FUNCTION_BLOCK basicFalhaFeedbackOnOff (* Basic Function Block Type *)
  (* Standard: 61499-2 *)
  (* Version 0.0, 1/26/2026, Schneider Electric, Template *)
  PACKAGE Hidryco.HidrycoLib;
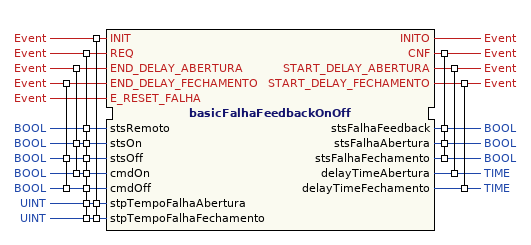
  EVENT_INPUT
    INIT WITH stpTempoFalhaAbertura, stpTempoFalhaFechamento; (* Initialization Request *)
    REQ WITH stsRemoto, stpTempoFalhaAbertura, stpTempoFalhaFechamento, stsOn, stsOff, cmdOn, cmdOff; (* Normal Execution Request *)
    END_DELAY_ABERTURA WITH stsOn, cmdOn;
    END_DELAY_FECHAMENTO WITH stsOff, cmdOff;
    E_RESET_FALHA;
  END_EVENT
  EVENT_OUTPUT
    INITO; (* Initialization Confirm *)
    CNF WITH stsFalhaFeedback, stsFalhaAbertura, stsFalhaFechamento; (* Execution Confirmation *)
    START_DELAY_ABERTURA WITH delayTimeAbertura;
    START_DELAY_FECHAMENTO WITH delayTimeFechamento;
  END_EVENT
  VAR_INPUT
    stsRemoto : BOOL;
    stsOn : BOOL;
    stsOff : BOOL;
    cmdOn : BOOL;
    cmdOff : BOOL;
    stpTempoFalhaAbertura : UINT;
    stpTempoFalhaFechamento : UINT;
  END_VAR
  VAR_OUTPUT
    stsFalhaFeedback : BOOL;
    stsFalhaAbertura : BOOL;
    stsFalhaFechamento : BOOL;
    delayTimeAbertura : TIME;
    delayTimeFechamento : TIME;
  END_VAR
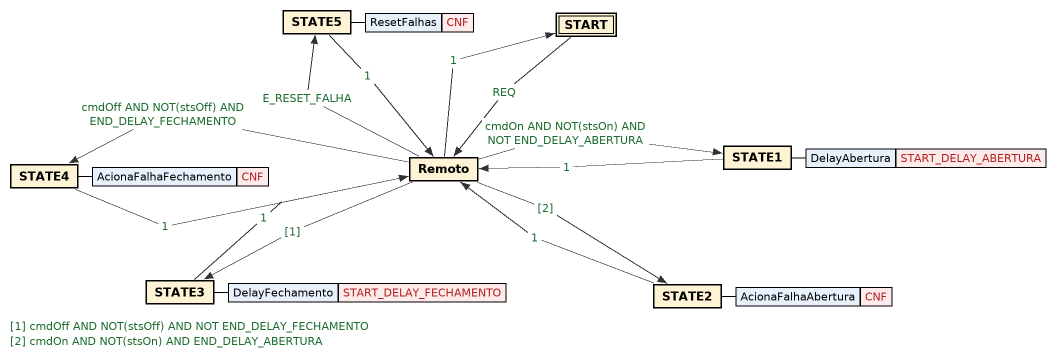
  EC_STATES
    START; (* Initial State *)
    Remoto;
    STATE1 : DelayAbertura -> START_DELAY_ABERTURA;
    STATE2 : AcionaFalhaAbertura -> CNF;
    STATE3 : DelayFechamento -> START_DELAY_FECHAMENTO;
    STATE4 : AcionaFalhaFechamento -> CNF;
    STATE5 : ResetFalhas -> CNF;
  END_STATES
  EC_TRANSITIONS
    START TO Remoto := REQ;
    Remoto TO STATE1 := cmdOn AND NOT(stsOn) AND NOT END_DELAY_ABERTURA;
    STATE1 TO Remoto := 1;
    Remoto TO STATE2 := cmdOn AND NOT(stsOn) AND END_DELAY_ABERTURA;
    STATE2 TO Remoto := 1;
    Remoto TO STATE3 := cmdOff AND NOT(stsOff) AND NOT END_DELAY_FECHAMENTO;
    STATE3 TO Remoto := 1;
    Remoto TO STATE4 := cmdOff AND NOT(stsOff) AND END_DELAY_FECHAMENTO;
    STATE4 TO Remoto := 1;
    Remoto TO STATE5 := E_RESET_FALHA;
    STATE5 TO Remoto := 1;
    Remoto TO START := 1;
  END_TRANSITIONS
  ALGORITHM INIT IN ST: (* Initialization algorithm *)
;
  END_ALGORITHM
  ALGORITHM REQ IN ST: (* Normally executed algorithm *)
;
  END_ALGORITHM
  ALGORITHM DelayAbertura IN ST:
delayTimeAbertura := DINT_TO_TIME(UINT_TO_DINT(stpTempoFalhaAbertura) * 1000);
;
  END_ALGORITHM
  ALGORITHM DelayFechamento IN ST:
delayTimeFechamento := DINT_TO_TIME(UINT_TO_DINT(stpTempoFalhaFechamento) * 1000);
;
  END_ALGORITHM
  ALGORITHM AcionaFalhaAbertura IN ST:
IF (cmdOn AND NOT(stsOn)) THEN
	stsFalhaAbertura := TRUE;
	stsFalhaFeedback := TRUE;
END_IF
;
  END_ALGORITHM
  ALGORITHM AcionaFalhaFechamento IN ST:
IF (cmdOff AND NOT(stsOff)) THEN
	stsFalhaFechamento := TRUE;
	stsFalhaFeedback := TRUE;
END_IF
;
  END_ALGORITHM
  ALGORITHM ResetFalhas IN ST:
stsFalhaAbertura := FALSE;
stsFalhaFechamento := FALSE;
stsFalhaFeedback := FALSE;
;
  END_ALGORITHM
END_FUNCTION_BLOCK
